RoboDK station: robotics_project 1626489.rdk

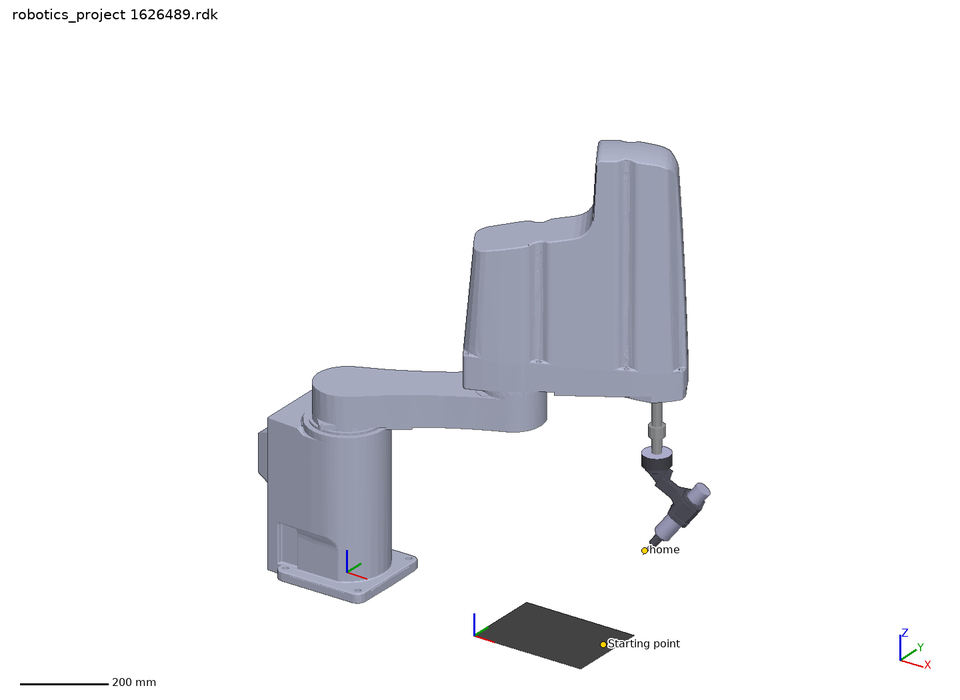
[picture v0: the station drawn from its stored meshes, robots at their saved joint values, targets as dots, program paths as lines]
Station robotics_project 1626489 (saved by RoboDK 5.3.2). Poses are relative to the parent item; angles as X-Y-Z fixed-axis rotations.
  - frame Mitsubishi RH-12FH7035 Base at (0, 0, 0) mm
    - robot Mitsubishi RH-12FH7035: 4 axes, payload 12 kg, reach 600 mm, repeatability 0.025 mm
        modified DH rows (alpha deg, a mm, theta deg, d mm): 0, 0, 0, 0; 0, 375, 0, 0; 0, 325, 0, 0 linear; 180, 0, 0, 0
        joint limits [-132, -150, 0, -360] to [132, 150, 300, 360]; home [0, 0, 350, 0]; saved at [32.01, 0, 300, -8.37]
      - tool Spindle, TCP at (-28, 0, -230) mm, rotated rx 0 ry 0 rz 10 deg, size 157.3 x 72 x 259.9 mm
  - Python program Prog1 (listed below)
  - frame Object frame at (396.57, -64.82, -22.29) mm
    - target Starting point (Cartesian target) at (265.37, 127.67, 1) mm, rotated rx 0 ry 0 rz -49.54 deg; joints [53.613, -106.441, 207.706, -6.712] of Mitsubishi RH-12FH7035
    - object A4 at (0, 0, 0) mm, size 297 x 210 x 1 mm, geometry from A4.STEP
    - target home (Cartesian target) at (171.35, 424.64, 92.29) mm, rotated rx 0 ry 0 rz 33.64 deg; joints [32.01, 0, 300, -8.37] of Mitsubishi RH-12FH7035

--- Python program Prog1 ---
from robolink import *    # RoboDK API
from robodk import *      # Robot toolbox

name_path = getOpenFile(r"C:\Users\alyaf\Desktop\myname.csv") #reading x, y &z from a csv file
name_list = LoadList(name_path) #storing the values in a matrix/list called (name_list)

RDK = Robolink()

robot = RDK.Item('',ITEM_TYPE_ROBOT)

home = RDK.Item('home') #Defining Home
O_frame = RDK.Item('Object frame') #Defining a frame for the A4 object
start_eng = RDK.Item('Starting point')#Defining a tareget to start engraving
target_pose = start_eng.Pose()


robot.setPoseFrame(O_frame)


#Drawing the full name around the reference target
for i in range(len(name_list)):
    a = target_pose
    a.setPos(name_list[i])
    start_eng.setPose(a)

    if i == 0:
        robot.MoveJ(start_eng)
    else:
        robot.MoveL(start_eng)




#return back to home
robot.MoveJ(home)
